TEXTLIST tlActualMachineName
  0 = 'Filler A - BA02PL01_M1'
  1 = 'Cork - BA02PL01_M2'
  2 = 'Filler B - BA02PL03'
  3 = 'Sticker - BA02PL06_M1'
  4 = 'Laser - BA02PL06_M2'
   = ''
END_TEXTLIST

(* stored: Version 1.1.0.1, ProductVersion 3.1.4024.13
   TextList tlActualMachineName: Id {3bd058b3-ac03-45e1-8314-b47637397e44} *)
